FUNCTION_BLOCK FB_LensSetCompounderMock EXTENDS FB_FalliblePublicMock IMPLEMENTS I_LensSetCompounder
VAR
    fbFocalLengthCompounded : FB_QuantityLREALPublic(Units := 'm');
    afFocalLength : ARRAY[1..GVL_Physics.nMaxNumLensesInSet] OF LREAL;
    nIndex : INT;
END_VAR


METHOD Compound
VAR_INPUT
    FocalLength : I_QuantityLREAL;
    SourceDistance : I_QuantityLREAL;
END_VAR
VAR_IN_OUT
    FocalLengthCompounded : FB_QuantityLREALPublic(Units := 'm');
END_VAR

FocalLengthCompounded := fbFocalLengthCompounded;
END_METHOD


METHOD Reset
END_METHOD


METHOD SetResult
VAR_INPUT
    Result : LREAL;
    LensNum : INT;
END_VAR

afFocalLength[LensNum] := Result;
END_METHOD


METHOD SetValid

fbFocalLengthCompounded.Val := 1.0;
fbFocalLengthCompounded.Units := 'm';
fbFocalLengthCompounded.ClearError();
ClearError();
END_METHOD

END_FUNCTION_BLOCK

(* stored: Version 1.1.0.1
   POU FB_LensSetCompounderMock: Id {67b527a3-9387-46bb-810d-7075318f36e8}, SpecialFunc None
   Method Compound: Id {75ebd25a-6006-41a6-afc8-68dd6ba211e1}
   Method Reset: Id {01cee560-272e-4fe8-acac-ea83151ba838}
   Method SetResult: Id {d3e63f9a-6509-4a0d-a4de-234257a7bd56}
   Method SetValid: Id {32c5277f-0827-4d86-91f4-c676cc2b02f3} *)
